Staubli VAL3: Queue.pjx

--- Queue.pjx ---
Parameters version=s7.7.2 stackSize=5000 millimeterUnit=true
Program file=start.pgx
Program file=stop.pgx
Data file=Queue.dtx
Type name=MotionCmd path=Disk://ros_libs/MotionCmd/MotionCmd.pjx

--- Queue.dtx ---
public num nPush
public num nPop
public num nElems
public MotionCmd buffer[10]
  [0]
    mdesc mDesc = {leave=0, reach=0}
    num nDuration
    num nSequence
    jointRx jJointRx
  [1]
    mdesc mDesc = {leave=0, reach=0}
    num nDuration
    num nSequence
    jointRx jJointRx
  [2]
    mdesc mDesc = {leave=0, reach=0}
    num nDuration
    num nSequence
    jointRx jJointRx
  [3]
    mdesc mDesc = {leave=0, reach=0}
    num nDuration
    num nSequence
    jointRx jJointRx
  [4]
    mdesc mDesc = {leave=0, reach=0}
    num nDuration
    num nSequence
    jointRx jJointRx
  [5]
    mdesc mDesc = {leave=0, reach=0}
    num nDuration
    num nSequence
    jointRx jJointRx
  [6]
    mdesc mDesc = {leave=0, reach=0}
    num nDuration
    num nSequence
    jointRx jJointRx
  [7]
    mdesc mDesc = {leave=0, reach=0}
    num nDuration
    num nSequence
    jointRx jJointRx
  [8]
    mdesc mDesc = {leave=0, reach=0}
    num nDuration
    num nSequence
    jointRx jJointRx
  [9]
    mdesc mDesc = {leave=0, reach=0}
    num nDuration
    num nSequence
    jointRx jJointRx

--- start.pgx ---
program start()
begin
  // Copyright (c) 2016, Ocado Technology - Robotics Research Team
  //
  // Licensed under the Apache License, Version 2.0 (the "License");
  // you may not use this file except in compliance with the License.
  // You may obtain a copy of the License at
  //
  //     http://www.apache.org/licenses/LICENSE-2.0
  //
  // Unless required by applicable law or agreed to in writing, software
  // distributed under the License is distributed on an "AS IS" BASIS,
  // WITHOUT WARRANTIES OR CONDITIONS OF ANY KIND, either express or implied.
  // See the License for the specific language governing permissions and
  // limitations under the License.



end
